// TIA Portal V15.1 export
// export: Created 2024-06-21T08:40:55.3925685Z, ExportSetting WithDefaults, DisplayName Totally Integrated Automation Portal, DisplayVersion V15.1 Update 5, DisplayName TIA Portal Openness, DisplayVersion V15.1 Update 5, DisplayName SINAMICS Startdrive Advanced, DisplayVersion V15.1, DisplayName G130, G150, S120, S150, SINAMICS MV, S210, DisplayVersion V15.1, DisplayName G110M, G120, G120C, G120D, G120P, DisplayVersion V15.1, DisplayName STEP 7 Professional, DisplayVersion V15.1 Update 5, DisplayName STEP 7 Safety, DisplayVersion V15.1, DisplayName WinCC Professional, DisplayVersion V15.1 Update 5, DisplayName SIMATIC Visualization Architect, DisplayVersion V15.1
FUNCTION "LIncInt" : Void   // FC2118, FBD
TITLE = LInc
{ S7_Optimized_Access := 'TRUE' }
AUTHOR : VCC
FAMILY : Control
VERSION : 0.1
// =============================================================================
// This Module Increase The Value With 1 Every Scan In IO_Inc
// =============================================================================
// stored: AutoNumber false, IsIECCheckEnabled true, SetENOAutomatically False, UDAEnableTagReadback false
   VAR_IN_OUT
      IO_INC : Int;   // Value
   END_VAR
BEGIN

NETWORK
TITLE = **** 4.4 - Machine status - Calculated **** Increment
// Increment
      L     #IO_INC;
      +     1;
      T     #IO_INC;
END_FUNCTION
